RoboDK station: Sini123456789.rdk

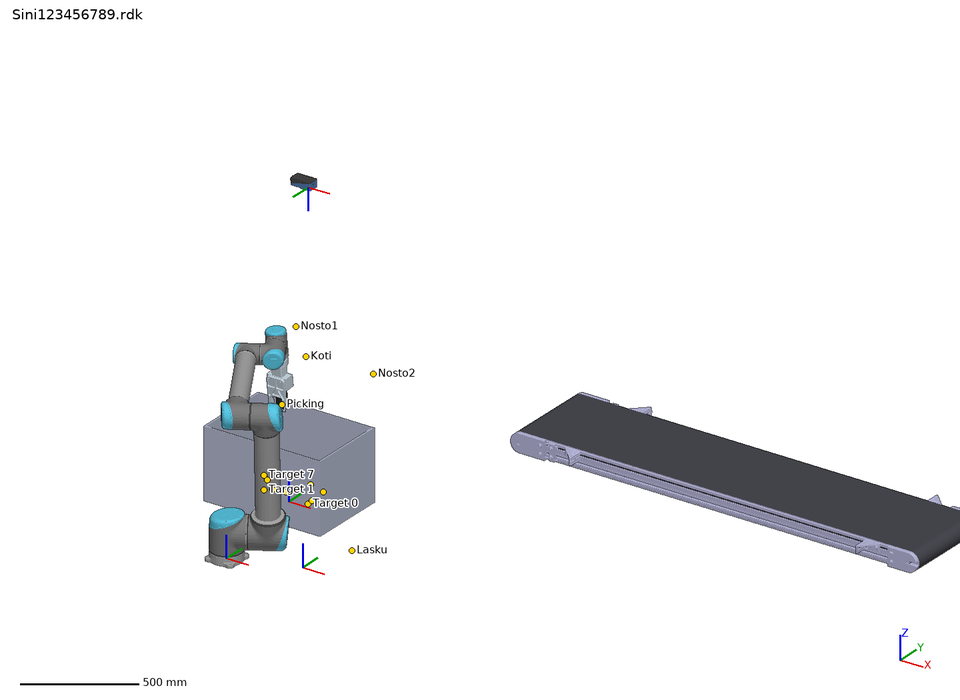
[picture v0: the station drawn from its stored meshes, robots at their saved joint values, targets as dots, program paths as lines]
Station Sini123456789. Poses are relative to the parent item; angles as X-Y-Z fixed-axis rotations.
  - frame LaatikonKoord at (-100, 600, 0) mm
    - object Laatikko at (0, 0, 0) mm, rotated rx 90 ry 0 rz 0 deg, size 600 x 350 x 400 mm, geometry from Laatikko.STEP
    - object Harjanvarsi at (0, 0, 0) mm, rotated rx 90 ry 0 rz 0 deg, size 30 x 30 x 325 mm, geometry from Harjanvarsi.STEP
    - object Harjanvarsi 0 at (92.45, 6.84, 10) mm, rotated rx 90 ry 0 rz 43.06 deg, size 30 x 30 x 325 mm, geometry from Harjanvarsi.STEP
    - target Target 0 (Cartesian target) at (92.45, 6.84, 10) mm, rotated rx 180 ry 0 rz -43.06 deg; joints [99.416, -92.641, -87.294, -0.065, 79.846, 0] of UR10
    - object Harjanvarsi 1 at (-124.07, -5.25, 20) mm, rotated rx 90 ry 0 rz 27.3 deg, size 30 x 30 x 325 mm, geometry from Harjanvarsi.STEP
    - target Target 1 (Cartesian target) at (-124.07, -5.25, 20) mm, rotated rx 180 ry 0 rz -27.3 deg; joints [99.416, -92.641, -87.294, -0.065, 79.846, 0] of UR10
    - object Harjanvarsi 2 at (-85.85, 4.75, 30) mm, rotated rx 90 ry 0 rz 37.73 deg, size 30 x 30 x 325 mm, geometry from Harjanvarsi.STEP
    - target Target 2 (Cartesian target) at (-85.85, 4.75, 30) mm, rotated rx 180 ry 0 rz -37.73 deg; joints [99.416, -92.641, -87.294, -0.065, 79.846, 0] of UR10
    - object Harjanvarsi 3 at (122.18, -6.06, 40) mm, rotated rx 90 ry 0 rz -51.16 deg, size 30 x 30 x 325 mm, geometry from Harjanvarsi.STEP
    - target Target 3 (Cartesian target) at (122.18, -6.06, 40) mm, rotated rx 180 ry 0 rz 51.16 deg; joints [99.416, -92.641, -87.294, -0.065, 79.846, 0] of UR10
    - object Harjanvarsi 4 at (-5.98, -15.09, 50) mm, rotated rx 90 ry 0 rz -43.34 deg, size 30 x 30 x 325 mm, geometry from Harjanvarsi.STEP
    - target Target 4 (Cartesian target) at (-5.98, -15.09, 50) mm, rotated rx 180 ry 0 rz 43.34 deg; joints [99.416, -92.641, -87.294, -0.065, 79.846, 0] of UR10
    - object Harjanvarsi 5 at (-122.82, 16.93, 60) mm, rotated rx 90 ry 0 rz 59.8 deg, size 30 x 30 x 325 mm, geometry from Harjanvarsi.STEP
    - target Target 5 (Cartesian target) at (-122.82, 16.93, 60) mm, rotated rx 180 ry 0 rz -59.8 deg; joints [99.416, -92.641, -87.294, -0.065, 79.846, 0] of UR10
    - object Harjanvarsi 6 at (55.67, -6.34, 70) mm, rotated rx 90 ry 0 rz -62.98 deg, size 30 x 30 x 325 mm, geometry from Harjanvarsi.STEP
    - target Target 6 (Cartesian target) at (55.67, -6.34, 70) mm, rotated rx 180 ry 0 rz 62.98 deg; joints [99.416, -92.641, -87.294, -0.065, 79.846, 0] of UR10
    - object Harjanvarsi 7 at (-135.04, 10.5, 80) mm, rotated rx 90 ry 0 rz 5.25 deg, size 30 x 30 x 325 mm, geometry from Harjanvarsi.STEP
    - target Target 7 (Cartesian target) at (-135.04, 10.5, 80) mm, rotated rx 180 ry 0 rz -5.25 deg; joints [99.416, -92.641, -87.294, -0.065, 79.846, 0] of UR10
    - object Harjanvarsi 8 at (172.56, 6.39, 90) mm, rotated rx 90 ry 0 rz 0.31 deg, size 30 x 30 x 325 mm, geometry from Harjanvarsi.STEP
    - target Target 8 (Cartesian target) at (172.56, 6.39, 90) mm, rotated rx 180 ry 0 rz -0.31 deg; joints [99.416, -92.641, -87.294, -0.065, 79.846, 0] of UR10
    - object Harjanvarsi 9 at (99.45, 19.22, 100) mm, rotated rx 90 ry 0 rz 24.91 deg, size 30 x 30 x 325 mm, geometry from Harjanvarsi.STEP
    - target Target 9 (Cartesian target) at (99.45, 19.22, 100) mm, rotated rx 180 ry 0 rz -24.91 deg; joints [99.416, -92.641, -87.294, -0.065, 79.846, 0] of UR10
  - frame Conveyor Belt Base at (547.04, -221.72, 200) mm
    - target Lasku (Cartesian target) at (100, 220, 20) mm, rotated rx 179.49 ry -0.51 rz -90.12 deg; joints [100, 0, 0, 0, 0, 0]
    - robot Conveyor Belt: 1 axes
        modified DH rows (alpha deg, a mm, theta deg, d mm): 0, 0, 0, 0 linear
        base shift (0, 0, 0) mm, rotated rx 0 ry 90 rz 0 deg
        joint limits [-500000] to [500000]; home [0]; saved at [0]
  - frame UR10 Base at (0, 0, 0) mm
    - robot UR10: 6 axes, payload 10 kg, reach 1300 mm, repeatability 0.1 mm, weight 28.9 kg
        modified DH rows (alpha deg, a mm, theta deg, d mm): 0, 0, 0, 128; 90, 0, 180, 0; 0, 612.7, 0, 0; 0, 571.6, 0, 163.9; -90, 0, 0, 115.7; 90, 0, 180, 92.2
        joint limits [-360, -360, -360, -360, -360, -360] to [360, 360, 360, 360, 360, 360]; home [0, -90, -90, 0, 90, 0]; saved at [120.399, -78.882, -99.842, -84.683, 86.032, 30.908]
      - tool Gripper, TCP at (0, 0, 233.37) mm, size 100 x 89.2 x 240.5 mm
    - target Koti (Cartesian target) at (167.76, 344.11, 856.4) mm, rotated rx -90 ry 0 rz -0.74 deg; joints [91.138, -35.831, -117.783, -26.385, 88.124, 0] of UR10
    - target Nosto1 (Cartesian target) at (-53.95, 587.76, 837.61) mm, rotated rx -134.04 ry 0 rz -13.2 deg; joints [132.49, -66.962, -79.737, -93.063, 53.572, 45.532] of UR10
    - target Nosto2 (Cartesian target) at (725.81, 39.42, 1052.1) mm, rotated rx -93.82 ry 0.09 rz -86.95 deg; joints [129.094, -64.812, -80.46, -91.092, 66.097, -1.606] of UR10
    - target Picking (Cartesian target) at (-145.61, 616.62, 432.57) mm, rotated rx -172.31 ry 0 rz -0.74 deg; joints [120.399, -78.882, -99.842, -84.683, 86.032, 30.908] of UR10
  - frame Kamera at (0, 600, 1500) mm, rotated rx 180 ry 0 rz 0 deg
    - object SICK VSPP-5f2113 at (0, 0, 0) mm, size 53 x 116 x 38 mm, geometry from Cam2D_SICK_VSPP_5F2113.sld
  - Python program KameranAvaaminen (listed below)
  - Python program KappaleenLuominenLaatikkoon (listed below)
  - Python program RobotinOhjaus (listed below)
  - Python program Siivous (listed below)
  - program Simulaatio (3 instructions, listed below)

--- Python program KameranAvaaminen ---
from robolink import *    # RoboDK API
from robodk import *      # Robot toolbox
RDK = Robolink()

RDK.Cam2D_Close()
camref = RDK.Item('Kamera',ITEM_TYPE_FRAME)

cam_id = RDK.Cam2D_Add(camref, 'FOCAL_LENGHT=17 FOV=32 FAR_LENGHT=1700 SIZE=640x480 BG_COLOR=black LIGHT_AMBIENT=white LIGHT_DIFFUSE=black LIGHT_SPECULAR=white')

--- Python program KappaleenLuominenLaatikkoon ---
# Type help("robolink") or help("robodk") for more information
# Press F5 to run the script
# Documentation: https://robodk.com/doc/en/RoboDK-API.html
# Reference:     https://robodk.com/doc/en/PythonAPI/index.html
# Note: It is not required to keep a copy of this file, your python script is saved with the station
from robolink import *    # RoboDK API
from robodk import *      # Robot toolbox
from random  import uniform
import time
RDK = Robolink()
count = 0
RandZ = 0


frame_Laatikko = RDK.Item('LaatikonKoord', ITEM_TYPE_FRAME)

varsi = RDK.Item('Harjanvarsi')
varsi.Copy()

while count < 10:
    newpart = frame_Laatikko.Paste()
    newpart.setName('Harjanvarsi '+str(count))

    RandX = uniform(-250, 250)
    RandY = uniform(-20, 20)
    RandZ += 10
    RotZ = uniform(-1.1, 1.1)

    newpart.setPose(TxyzRxyz_2_Pose([RandX,RandY,RandZ,1.5708,RotZ,0]))
    newpart.setVisible(True, False)

    target = RDK.AddTarget("Target "+str(count), frame_Laatikko)
    target.setPose(TxyzRxyz_2_Pose([RandX,RandY,RandZ,3.14159,0,RotZ]))

    count += 1

--- Python program RobotinOhjaus ---
from robolink import *    # RoboDK API
from robodk import *      # Robot toolbox
import time
RDK = Robolink()

Robot = RDK.Item('UR10', ITEM_TYPE_ROBOT)
Tool = RDK.Item('Gripper', ITEM_TYPE_TOOL)

Koti  = RDK.Item('Koti')
Picking = RDK.Item('Picking')
Nosto1  = RDK.Item('Nosto1')
Nosto2  = RDK.Item('Nosto2')
Lasku  = RDK.Item('Lasku')

frame_Robot = RDK.Item('UR10 Base', ITEM_TYPE_FRAME)
frame_Laatikko = RDK.Item('LaatikonKoord', ITEM_TYPE_FRAME)
frame_Kuljetin = RDK.Item('Conveyor Belt Base', ITEM_TYPE_FRAME)

Approach = 50
count = 19

def TCP_On(toolitem):
    """Attaches the closest object to the toolitem Htool pose,
    It will also output appropriate function calls on the generated robot program (call to TCP_On)"""
    toolitem.AttachClosest()
    toolitem.RDK().RunMessage('Set air valve on')
    toolitem.RDK().RunProgram('TCP_On()');



def TCP_Off(toolitem, itemleave=0):
    """Detaches the closest object attached to the toolitem Htool pose,
    It will also output appropriate function calls on the generated robot program (call to TCP_Off)"""
    toolitem.DetachAll(itemleave)
    toolitem.RDK().RunMessage('Set air valve off')
    toolitem.RDK().RunProgram('TCP_Off()');

harjat = []

"""def add(objects, startswith="Harjanvarsi "):
#Poistaa kaikki esineet, joiden nimi alkaa "Harjanvarsi".
    for item in objects:
        if item.Name().startswith(startswith):
            item.Copy()
            item.Paste


all_objects = RDK.ItemList(ITEM_TYPE_OBJECT, False)
add(all_objects, 'Harjanvarsi ')

harjat = RDK.ItemList(ITEM_TYPE_OBJECT, False)

n = len(harjat)
print (n)
n -= 1
print (n)
Robot.setPoseTool(Tool) """

n = 9
while count > 0:
    #print (all_objects[n])
    Robot.MoveJ(Koti)
    Robot.MoveJ(Picking)

    #part_position_i = all_objects[n]

    time.sleep(2)

    Robot.setPoseFrame(frame_Laatikko)
    Target = RDK.Item('Target '+str(count))
    Robot.MoveJ(Target)
    TCP_On(Tool)

    Robot.setPoseFrame(frame_Robot)
    Robot.MoveJ(Nosto1)
    Robot.MoveJ(Nosto2)

    Robot.setPoseFrame(frame_Kuljetin)
    Robot.MoveJ(Lasku)
    TCP_Off(Tool, frame_Kuljetin)
    Robot.setPoseFrame(frame_Robot)

    n -= 1

Robot.MoveJ(Koti)

--- Python program Siivous ---
from robolink import *    # RoboDK API
from robodk import *      # Robot toolbox
RDK = Robolink()


#Siivotaan aikaisemmin luodut Objectit

def cleanup(objects, startswith="Harjanvarsi "):
#Poistaa kaikki esineet, joiden nimi alkaa "Harjanvarsi".
    for item in objects:
        if item.Name().startswith(startswith):
            item.Delete()


all_objects = RDK.ItemList(ITEM_TYPE_OBJECT, False)
cleanup(all_objects, 'Harjanvarsi ')

all_targets = RDK.ItemList(ITEM_TYPE_TARGET, False)
cleanup(all_targets, 'Target')

--- program Simulaatio (robot UR10) ---
  Call KameranAvaaminen
  Call KappaleenLuominenLaatik...: KappaleenLuominenLaatikkoon
  Call RobotinOhjaus
